TYPE WcStateBase_A2171C4E :
STRUCT
END_STRUCT
END_TYPE

(* stored: Version 1.2.0.0, ProductVersion 3.1.4024.9
   DUT WcStateBase_A2171C4E: Id {40e796e6-a83e-423a-8722-392e2863156e} *)
